// TIA Portal V17 export
// export: Created 2021-12-03T08:13:12.1129913Z, ExportSetting WithDefaults, DisplayName Totally Integrated Automation Portal, DisplayVersion V17, DisplayName TIA Portal Openness, DisplayVersion V17, DisplayName TIA Portal Version Control Interface, DisplayVersion V17, DisplayName STEP 7 Professional, DisplayVersion V17, DisplayName STEP 7 Safety, DisplayVersion V17, DisplayName WinCC Advanced, DisplayVersion V17
DATA_BLOCK "FGDB_ContCtrl"   // DB700, F_DB
VERSION : 0.1
// stored: AutoNumber false
   VAR
      ModCont400_Rel : Bool;   // Modulator: Contactor 400VAC - Release / Разрешение включения контактора модулятора 3 фазы / Разрешение включения модулятора 400 В
      ModCont230_Rel : Bool;   // Modulator: Contactor 230VAC - Release / Разрешение включения контактора модулятора 1 фаза / Разрешение включения модулятора 230 В
      ChilCont_Rel : Bool;   // Chiller: Contactor - Release / Разрешение включения контактора чиллера / Разрешение включения чиллера
      AccCont_Rel : Bool;   // Разрешение включения консоли ускорителя / Разрешение включения ускорителя
      ModCont400_Err : Bool;   // Ошибка при включении модулятора 400В
      ModCont230_Err : Bool;   // Ошибка при включении модулятора 230В
      ChillCont_Err : Bool;   // Ошибка при включении чиллера
      AccCont_Err : Bool;   // Ошибка при включении ускорителя
      ModCont400_AckReq : Bool;   // Готовность к сбросу при включении модулятора 400В
      ModCont230_AckReq : Bool;   // Готовность к сбросу при включении модулятора 230В
      ChillCont_AckReq : Bool;   // Готовность к сбросу при включении чиллера
      AccCont_AckReq : Bool;   // Готовность к сбросу при включении ускорителя
      ChilOff_DlyTm : Time;   // Время выключения
      ChilOn_DlyTm : Time;   // Время включения
      ChilCont_OfTof : Bool;
      ChilCont_OfIn : Bool;
      ChilCont_OnTon : Bool;
      Mod400_OnDly : Bool;   // Задержка между включением 230 и 380 В
      "X-RayOn" : Bool;
      ConvCont_Rel : Bool;   // Разрешение включения контактора
      ConvCont_Err : Bool;
      ConvCont_AckReq : Bool;
   END_VAR
BEGIN
END_DATA_BLOCK
